FUNCTION_BLOCK FB_PMLStateMachine_Tests EXTENDS FB_TestSuite
VAR
	PackMLStateMachine : PMLStateMAchine;
	TestSuiteTimer : TON := (PT := T#1S);
END_VAR

SetInitialModeForStateMachine();
AbortStateMachineFromUndefined();
SetStateCompleteTest();

PackMLStateMachine();

METHOD AbortStateMachineFromUndefined
VAR
	currentState : E_PMLState;
END_VAR
IF TEST_ORDERED('AbortStateMachineFromUndefined') THEN
	IF TestSuiteTimer.IN THEN
		PackMLStateMachine.PmlStateCommand(Command := E_PMLCommand.ePMLCommand_Abort);
		currentState := PackMLStateMachine.GetCurrentState();
		
		IF TestSuiteTimer.Q THEN
			AssertEquals_UDINT(Expected := E_PMLState.ePMLState_Aborting,
								Actual := currentState,
								Message := 'State machine didnt go into aborting');
			TestSuiteTimer(in := FALSE);
			TEST_FINISHED();
		END_IF
	ELSE
		currentState := PackMLStateMachine.GetCurrentState();
		AssertEquals_UDINT(Expected := E_PMLState.ePMLState_Undefined,
						Actual := currentState,
						Message := 'State machine not in undefined');
	END_IF
	
	
	TestSuiteTimer(IN := TRUE);
END_IF
END_METHOD

METHOD Register3SubUnits
VAR
	subUnit1 : PMLStateMachine;
	subUnit2 : PMLStateMachine;
	subUnit3 : PMLStateMachine;
	
	bOK : BOOL;
	numberOfSubUnits : INT;
END_VAR
IF TEST_ORDERED('Register3SubUnits') THEN

bOK := PackMLStateMachine.RegisterSubUnit(SubUnit := subUnit1 );
AssertTrue(Condition := bOK, Message := 'Subunit not added');	
numberOfSubUnits := PackMLStateMachine.GetNumberOfSubUnits;
AssertEquals_INT(Expected := 1, 
					Actual := numberOfSubUnits, 
					Message := 'Expected one event');

bOK := PackMLStateMachine.RegisterSubUnit(SubUnit := subUnit2 );
AssertTrue(Condition := bOK, Message := 'Subunit not added');	
numberOfSubUnits := PackMLStateMachine.GetNumberOfSubUnits;
AssertEquals_INT(Expected := 2, 
					Actual := numberOfSubUnits, 
					Message := 'Expected two events');
					
bOK := PackMLStateMachine.RegisterSubUnit(SubUnit := subUnit3 );
AssertTrue(Condition := bOK, Message := 'Subunit not added');	
numberOfSubUnits := PackMLStateMachine.GetNumberOfSubUnits;
AssertEquals_INT(Expected := 3, 
					Actual := numberOfSubUnits, 
					Message := 'Expected three events');

END_IF
END_METHOD

METHOD SetInitialModeForStateMachine
VAR
	currentMode : DINT;
END_VAR
IF TEST_ORDERED('SetInitialModeForStateMachine') THEN
	IF TestSuiteTimer.IN THEN
		PackMLStateMachine.PmlModeCommand(Mode := E_PMLProtectedUnitMode.ePMLProtUnitMode_Production);
		currentMode := PackMLStateMachine.GetCurrentMode();
		
		IF TestSuiteTimer.Q THEN
			AssertEquals_DINT(Expected := E_PMLProtectedUnitMode.ePMLProtUnitMode_Production,
								Actual := currentMode,
								Message := 'State machine mode didnt go into production');
			TestSuiteTimer(IN := FALSE);			
			TEST_FINISHED();
		END_IF
	ELSE
		currentMode := PackMLStateMachine.GetCurrentMode();
		AssertEquals_DINT(Expected := E_PMLProtectedUnitMode.ePMLProtUnitMode_Invalid,
					Actual := currentMode,
					Message := 'State machine has a mode');
	END_IF
	
	
	TestSuiteTimer(IN := TRUE);
END_IF
END_METHOD

METHOD SetStateCompleteTest
VAR
	currentState : E_PMLState;
END_VAR
IF TEST_ORDERED('SetStateCompleteTest') THEN
	IF TestSuiteTimer.IN THEN
		PackMLStateMachine.SetStateComplete();
		currentState := PackMLStateMachine.GetCurrentState();
		
		IF TestSuiteTimer.Q THEN
			AssertEquals_UDINT(Expected := E_PMLState.ePMLState_Aborted,
								Actual := currentState,
								Message := 'State machine didnt go into Aborted');
			TestSuiteTimer(in := FALSE);
			TEST_FINISHED();
		END_IF
	ELSE
		currentState := PackMLStateMachine.GetCurrentState();
		AssertEquals_UDINT(Expected := E_PMLState.ePMLState_Aborting,
						Actual := currentState,
						Message := 'State machine not in aborting');
	END_IF
	
	
	TestSuiteTimer(IN := TRUE);
END_IF
END_METHOD

END_FUNCTION_BLOCK

(* stored: Version 1.1.0.1, ProductVersion 3.1.4024.11
   POU FB_PMLStateMachine_Tests: Id {153e17aa-3c02-42b4-9409-4e339c7b2e61}, SpecialFunc None
   Method AbortStateMachineFromUndefined: Id {be97a7d9-c1e6-47fd-868f-9e0735123da9}
   Method Register3SubUnits: Id {44486354-59f9-4c2f-be74-f3c1103bad46}
   Method SetInitialModeForStateMachine: Id {6edf451a-0e29-4c4b-abba-a91a12034924}
   Method SetStateCompleteTest: Id {7a62278c-da95-418c-a0e1-bdec97969de9} *)
